// TIA Portal V20 export
TYPE "LER_SignalsInput"
// stored: Access Published
   STRUCT
      ButtonLeft : Array[0..15] of Bool;
      ButtonRight : Array[0..15] of Bool;
   END_STRUCT;
END_TYPE
